{attribute 'pack_mode' := '1'}
TYPE TStickData :
STRUCT
	iBarrelPos			: INT := -1;
	lrDiameter			: LREAL;
	lrOutLength			: LREAL;
	lrTotalLength			: LREAL;
END_STRUCT
END_TYPE

(* stored: Version 1.1.0.1, ProductVersion 3.1.4022.12
   DUT TStickData: Id {694e4e59-b247-4190-a3ad-8e7086ee393f} *)
